{attribute 'GeneratedUsingTerminal: EK1960-2600-0021'}
{attribute addProperty BoxType "EK1960-2600-0021"}
{attribute addProperty Id "FSOEAT %Q*FSOE_CDFABDDF56"}
{attribute addProperty CRC "937346404"}
{attribute addProperty Size "56"}
TYPE FSoE_Outputs_37DEC564 :
STRUCT
	{attribute addProperty Name "FSOE"}
	FSOE AT %Q* : FSOE_CDFABDDF;
END_STRUCT
END_TYPE

(* stored: Version 1.2.0.0, ProductVersion 3.1.4024.9
   DUT FSoE_Outputs_37DEC564: Id {693f104f-ffe3-4839-9e31-9f9f7b0be1a8} *)
